// TIA Portal V17 export
// export: Created 2024-09-02T12:50:16.7458Z, ExportSetting WithDefaults, DisplayName Totally Integrated Automation Portal, DisplayVersion V17, DisplayName TIA Portal Openness, DisplayVersion V17, DisplayName TIA Portal Version Control Interface, DisplayVersion V17, DisplayName STEP 7 Professional, DisplayVersion V17, DisplayName STEP 7 Safety, DisplayVersion V17, DisplayName WinCC Professional, DisplayVersion V17
DATA_BLOCK "AnwDB_HMI_ScreenCall_OP70"   // DB258
{ S7_Optimized_Access := 'TRUE'; DB_Accessible_From_OPC_UA := 'FALSE' }
AUTHOR : OlegFuehrus
FAMILY : HMI
NAME : HMI
VERSION : 0.1
// stored: AutoNumber true, DBAccessibleFromOPCUA false, IsOnlyStoredInLoadMemory false, IsRetainMemResEnabled false, IsWriteProtectedInAS false, MemoryReserve 100
   VAR
      ScreenNrCurrent : Int;   // Bildnummer aktuell / Current image number
      ScreenNrOld : Int;   // Bildnummer alt / Picture number old
      EdgeScreenChange : Bool;
      "ScreenCall[0]" : Array[1..16] of Struct
         HM : Bool;
         "Time" { S7_SetPoint := 'True'} : TON_TIME;
      END_STRUCT;
      "ScreenCall[1]" : Array[1..16] of Struct
         HM : Bool;
         "Time" { S7_SetPoint := 'True'} : TON_TIME;
      END_STRUCT;
      HMI_Layout { S7_SetPoint := 'True'} : "type_HMI_Layout";
      ScreenFunctionsGroup : Array[0..11] of Int;
   END_VAR
BEGIN
END_DATA_BLOCK
